Fanuc KAREL source: KT00949.KL

PROGRAM KT00949
%NOLOCKGROUP
VAR
  ENTRY: INTEGER
  PNAME: STRING[80]
  VNAME: STRING[80]
  STATUS: INTEGER
  VALUE: ARRAY[4] OF BYTE
BEGIN
  ENTRY = 0
  PNAME = ''
  VNAME = 'VALUE'
  GET_VAR(ENTRY, PNAME, VNAME, VALUE, STATUS)
END KT00949
